// ---- POUs/Vorlagen/RFID/FB_RFID.TcPOU
FUNCTION_BLOCK FB_RFID
VAR_INPUT
	PermissionHardware	:	BOOL;	//Freigabe Hardware
	QuitError	:	BOOL;	//Fehler quittieren
	Reset	:	BOOL;	//Reset Commands
	SensorPartDetected	:	BOOL;	//Sensor Teil erkannt
	CommandID	:	WORD;	//Wird nach einem Befehl immer um 1 erhoeht
	ReadData	:	WORD;	//Gelesener Wert an der Stelle vom MemoryIndex
	Status	:	WORD;	//Status ungleich 0 = Fehler
	ActorInstanceIndex	:	INT;	//Index in DropDown HMI
	ActorInstanceName	:	STRING;		//Name of the instance
END_VAR
VAR_OUTPUT
	ExecuteCommand	:	BOOL;
	FMReadingSerialNumber	:	BOOL;	//Fertigmeldung Lesen Seriennummer
	FMReadingData	:	BOOL;	//Fertigmeldung Lesen
	FMWritingData	:	BOOL;	//Fertigmeldung Schreiben
	Error	:	BOOL;	//Fehler
	ErrorID	:	WORD;	//Fehler-ID
	Command	:	WORD;	//Command-ID:
	WriteData	:	WORD;	//Daten die geschrieben werden
	MemoryIndex	:	WORD;	//Angewaehlten Memory-Index der gelesen/geschrieben werden soll
	ReadDataTag	:	ARRAY[0..127] OF WORD;	//Array mit allen gelesenen Daten
END_VAR
VAR_IN_OUT
	HMIInterface	:	MachineSectionHMIInterface;	//HMI-Interface
END_VAR
VAR
	statReadingSerialNumber	:	BOOL;
	statExecuteCommand	:	BOOL;
	statReadingData	:	BOOL;
	statWritingData	:	BOOL;
	statErrorActive	:	BOOL;
	statReadingSerialnumberFinished	:	BOOL;
	statReadingDataFinished	:	BOOL;
	statWritingDataFinished	:	BOOL;
	statSelectedCommand	:	WORD;
	statErrorID	:	WORD;
	statLastCommandID	:	WORD;
	statReadSerialNumber	:	WORD;
	statDataToWrite	:	WORD;
	statSelectedMemoryIndex	:	WORD;
	statReadDataCompelete	:	ARRAY[0..127] OF WORD;
	statCompleteDataToWrite	:	ARRAY[0..127] OF WORD;
	statStateReadSerialNumber	:	RFIDReadSerialnumberStates;
	statStateWriteData	:	RFIDReadWriteDataStates;
	statStateReadData	:	RFIDReadWriteDataStates;
	statRisingEdgeNewOrder	:	R_TRIG;
	statTONDelayWritting	:	TON;
	statTONDelayReading	:	TON;
	debugStepMemory	:	INT;
	
	internHMIInterface	:	MachineSectionHMIInterface;
	internRisingEdgeExecuteCommand	:	R_TRIG;
	internRisingEdgeReadAllDataFinished	:	R_TRIG;
END_VAR
VAR CONSTANT
	NOCOMMAND	:	WORD := 0;
	READSERIALNUMBERCOMMAND	:	WORD := 1;
	READDATACOMMAND	:	WORD := 2;
	WRITEDATACOMMAND	:	WORD := 3;
	CLEARALLDATACOMMAND	:	WORD := 4;
END_VAR

(*===================== HMI INTERFACE =====================*)
internHMIInterface := HMIInterface;

IF internHMIInterface.ActiveMachineSection = MachineSection.RFID AND
	internHMIInterface.SelectedActor = ActorInstanceIndex THEN
	(*===================== Status-Interface =====================*)
	internHMIInterface.RFID.RFIDStatus.PermissionHardware := PermissionHardware;
	internHMIInterface.RFID.RFIDStatus.PartPresent := SensorPartDetected;
	internHMIInterface.RFID.RFIDStatus.ErrorActive := statErrorActive;
	internHMIInterface.RFID.RFIDStatus.FMReading := statReadingDataFinished OR statReadingSerialnumberFinished;
	internHMIInterface.RFID.RFIDStatus.FMWritting := statWritingDataFinished;
	(*===================== Data-Interface =====================*)
	internHMIInterface.RFID.RFIDData.AllReadData := statReadDataCompelete; 
	IF internRisingEdgeReadAllDataFinished.Q THEN
		internHMIInterface.RFID.RFIDData.AllWriteData := statReadDataCompelete;
	END_IF
	(*===================== Execute Command =====================*)
	internRisingEdgeExecuteCommand(CLK := internHMIInterface.RFID.RFIDControl.ExecuteCommand);
	IF internRisingEdgeExecuteCommand.Q THEN
		CASE internHMIInterface.RFID.RFIDControl.SelectedCommand OF
			NOCOMMAND :
				statReadingSerialNumber := FALSE;
				statReadingData := FALSE;
				statWritingData := FALSE;
			READSERIALNUMBERCOMMAND:
				statReadingSerialNumber := TRUE;
			READDATACOMMAND:
				statReadingData := TRUE;
			WRITEDATACOMMAND:
				statCompleteDataToWrite := internHMIInterface.RFID.RFIDData.AllWriteData;
				statWritingData := TRUE;	
		END_CASE
	END_IF
	
	(*===================== Write Interface =====================*)
	HMIInterface := internHMIInterface;
END_IF

(*===================== Error Handling =====================*)
IF QuitError AND statErrorActive THEN
	statErrorActive := FALSE;
	statErrorID := 0;
END_IF
IF Status <> 0 THEN
	statErrorActive := TRUE;
	statErrorID := Status;
END_IF
IF PermissionHardware AND SensorPartDetected THEN
	(*===================== Reset Data =====================*)
	statRisingEdgeNewOrder(CLK:= statReadingSerialNumber OR statReadingData OR 
								 statWritingData);
	IF NOT SensorPartDetected OR statRisingEdgeNewOrder.Q
	THEN
		ResetData_On();
	ELSIF Reset THEN
		ResetData_On();
		statSelectedCommand := NOCOMMAND;
		statStateReadSerialNumber := RFIDReadSerialnumberStates.WAITINGTRIGGER;	
		statStateWriteData := RFIDReadWriteDataStates.WAITINGTRIGGER;
	END_IF
	IF CommandID = 0 AND statLastCommandID <> 0 THEN
		statLastCommandID := 0;
	END_IF
	(*===================== Read Serialnumber =====================*)
	CASE statStateReadSerialNumber OF
		RFIDReadSerialnumberStates.WAITINGTRIGGER :
		debugStepMemory := RFIDReadSerialnumberStates.WAITINGTRIGGER;
			IF statReadingSerialNumber THEN
				statReadingSerialNumber := FALSE;
				statStateReadSerialNumber := RFIDReadSerialnumberStates.SETTRIGGER;
			END_IF
		RFIDReadSerialnumberStates.SETTRIGGER:
			debugStepMemory := RFIDReadSerialnumberStates.SETTRIGGER;
			statExecuteCommand := TRUE;
			statSelectedCommand := READSERIALNUMBERCOMMAND;
			statStateReadSerialNumber := RFIDReadSerialnumberStates.WAITINGRESPONSE;
		RFIDReadSerialnumberStates.WAITINGRESPONSE:
			debugStepMemory := RFIDReadSerialnumberStates.WAITINGRESPONSE;
			IF statErrorActive THEN
				statStateReadSerialNumber := RFIDReadSerialnumberStates.ERRORACTIVE;
			ELSIF CommandID <> statLastCommandID THEN
				statStateReadSerialNumber := RFIDReadSerialnumberStates.RESPONSE;
				statExecuteCommand := FALSE;
				statSelectedCommand := NOCOMMAND;
			END_IF
		RFIDReadSerialnumberStates.RESPONSE:
			debugStepMemory := RFIDReadSerialnumberStates.RESPONSE;
			statReadSerialNumber := ReadData;
			statReadingSerialnumberFinished := TRUE;
			statStateReadSerialNumber := RFIDReadSerialnumberStates.WAITINGTRIGGER;
		RFIDReadSerialnumberStates.ERRORACTIVE:
			debugStepMemory := RFIDReadSerialnumberStates.ERRORACTIVE;
			IF NOT statErrorActive THEN
				statStateReadSerialNumber := RFIDReadSerialnumberStates.WAITINGTRIGGER;
			END_IF
	END_CASE;
	(*===================== Read Data =====================*)
	statTONDelayReading(IN:= statStateReadData = RFIDReadWriteDataStates.SETTRIGGER, 
						 PT:= T#100MS);
	CASE statStateReadData OF
		RFIDReadWriteDataStates.WAITINGTRIGGER :
		debugStepMemory := RFIDReadWriteDataStates.WAITINGTRIGGER;
			IF statReadingData THEN
				statReadingData := FALSE;
				statSelectedCommand := READDATACOMMAND;
				statSelectedMemoryIndex := 1;
				statStateReadData := RFIDReadWriteDataStates.SETTRIGGER;
			END_IF
		RFIDReadWriteDataStates.SETTRIGGER:
			debugStepMemory := RFIDReadWriteDataStates.SETTRIGGER;
			IF statTONDelayReading.Q THEN
				statExecuteCommand := TRUE;
				statStateReadData := RFIDReadWriteDataStates.WAITINGRESPONSE;
			END_IF
		RFIDReadWriteDataStates.WAITINGRESPONSE:
			debugStepMemory := RFIDReadWriteDataStates.WAITINGRESPONSE;
			IF statErrorActive THEN
				statStateReadData := RFIDReadWriteDataStates.ERRORACTIVE;
			ELSIF CommandID <> statLastCommandID THEN
				statStateReadData := RFIDReadWriteDataStates.RESPONSE;
 				statExecuteCommand := FALSE;
			END_IF
		RFIDReadWriteDataStates.RESPONSE:
			debugStepMemory := RFIDReadWriteDataStates.RESPONSE;
			statReadDataCompelete[statSelectedMemoryIndex -1] := ReadData;
			IF statSelectedMemoryIndex >= 127 THEN
				statStateReadData := RFIDReadWriteDataStates.FINISHED;	
			ELSE
				statSelectedMemoryIndex := statSelectedMemoryIndex + 1;
				statStateReadData := RFIDReadWriteDataStates.SETTRIGGER;	
			END_IF
		RFIDReadWriteDataStates.ERRORACTIVE:
			debugStepMemory := RFIDReadWriteDataStates.ERRORACTIVE;
			IF NOT statErrorActive THEN
				statStateReadData := RFIDReadWriteDataStates.WAITINGTRIGGER;
			END_IF
		RFIDReadWriteDataStates.FINISHED:
			statReadingDataFinished := TRUE;
			statSelectedCommand := NOCOMMAND;
			statStateReadData := RFIDReadWriteDataStates.WAITINGTRIGGER;
	END_CASE;
	internRisingEdgeReadAllDataFinished(CLK := statReadingDataFinished);
	(*===================== Write Data =====================*)
	statTONDelayWritting(IN:= statStateWriteData = RFIDReadWriteDataStates.SETTRIGGER, 
						 PT:= T#100MS);
	CASE statStateWriteData OF
		RFIDReadWriteDataStates.WAITINGTRIGGER :
		debugStepMemory := RFIDReadWriteDataStates.WAITINGTRIGGER;
			IF statWritingData THEN
				statWritingData := FALSE;
				statSelectedCommand := WRITEDATACOMMAND;
				statSelectedMemoryIndex := 1;
				statStateWriteData := RFIDReadWriteDataStates.SETTRIGGER;
			END_IF
		RFIDReadWriteDataStates.SETTRIGGER:
			debugStepMemory := RFIDReadWriteDataStates.SETTRIGGER;
			IF statTONDelayWritting.Q THEN
				statExecuteCommand := TRUE;
				statDataToWrite := statCompleteDataToWrite[statSelectedMemoryIndex - 1];
				statStateWriteData := RFIDReadWriteDataStates.WAITINGRESPONSE;
			END_IF
		RFIDReadWriteDataStates.WAITINGRESPONSE:
			debugStepMemory := RFIDReadWriteDataStates.WAITINGRESPONSE;
			IF statErrorActive THEN
				statStateWriteData := RFIDReadWriteDataStates.ERRORACTIVE;
			ELSIF CommandID <> statLastCommandID THEN
				statStateWriteData := RFIDReadWriteDataStates.RESPONSE;
 				statExecuteCommand := FALSE;
			END_IF
		RFIDReadWriteDataStates.RESPONSE:
			debugStepMemory := RFIDReadWriteDataStates.RESPONSE;
			IF statSelectedMemoryIndex >= 127 THEN
				statStateWriteData := RFIDReadWriteDataStates.FINISHED;	
			ELSE
				statSelectedMemoryIndex := statSelectedMemoryIndex + 1;
				statStateWriteData := RFIDReadWriteDataStates.SETTRIGGER;	
			END_IF
		RFIDReadWriteDataStates.ERRORACTIVE:
			debugStepMemory := RFIDReadWriteDataStates.ERRORACTIVE;
			IF NOT statErrorActive THEN
				statStateWriteData := RFIDReadWriteDataStates.WAITINGTRIGGER;
			END_IF
		RFIDReadWriteDataStates.FINISHED:
			statWritingDataFinished := TRUE;
			statSelectedCommand := NOCOMMAND;
			statStateWriteData := RFIDReadWriteDataStates.WAITINGTRIGGER;
	END_CASE;
	(*===================== Save Data =====================*)
	statLastCommandID := CommandID;
ELSE
	statReadingSerialNumber := FALSE;	
	statReadingData := FALSE;
	statWritingData := FALSE;
	statExecuteCommand := FALSE;
	statReadingSerialnumberFinished := FALSE;
	statReadingDataFinished := FALSE;
	statWritingDataFinished := FALSE;
	statSelectedCommand := NOCOMMAND;
END_IF
(*===================== Outputs =====================*)
ExecuteCommand := statExecuteCommand;
FMReadingSerialNumber := statReadingSerialnumberFinished;
FMReadingData := statReadingDataFinished;
FMWritingData := statWritingDataFinished;
Error := statErrorActive;
ErrorID := statErrorID;
Command := statSelectedCommand;
WriteData := statDataToWrite;
MemoryIndex := statSelectedMemoryIndex;
ReadDataTag := statReadDataCompelete;

METHOD PUBLIC ReadDataComplete : BOOL
VAR_INPUT
	StartReadData	:	BOOL;
END_VAR
IF StartReadData THEN
	statReadingData := TRUE;
	ReadDataComplete := TRUE;
ELSE
	ReadDataComplete := FALSE;
END_IF
END_METHOD

METHOD PUBLIC ReadSerialNumber : BOOL
VAR_INPUT
	Start_ReadingSerialNumebr	:	BOOL;
END_VAR
IF Start_ReadingSerialNumebr AND NOT statErrorActive AND
	SensorPartDetected
THEN
	statReadingSerialNumber := TRUE;
	ReadSerialNumber := TRUE;
ELSE
	ReadSerialNumber := FALSE;			
END_IF
END_METHOD

METHOD PRIVATE ResetData_On : BOOL
VAR
	i :	INT;	//Laufvariable abloeschen gelesene Daten
END_VAR
statReadingSerialnumberFinished := FALSE;
statReadingDataFinished := FALSE;
statWritingDataFinished := FALSE;
statExecuteCommand := FALSE;
statReadSerialNumber := 0;
statDataToWrite := 0;
statSelectedMemoryIndex := 0;
statSelectedCommand := NOCOMMAND;
FOR i := 0 TO 127 DO
	statReadDataCompelete[i] := 0;
END_FOR

ResetData_On := TRUE;
END_METHOD

METHOD WriteDataComplete : BOOL
VAR_INPUT
	StartWriteData	:	BOOL;
	CompleteDataToWrite	:	ARRAY [0..127] OF WORD;
END_VAR
IF StartWriteData THEN
	statWritingData := TRUE;
	statCompleteDataToWrite := CompleteDataToWrite;	
	WriteDataComplete := TRUE;
ELSE
	WriteDataComplete := FALSE;
END_IF
END_METHOD

END_FUNCTION_BLOCK

// ---- POUs/Vorlagen/VisionSensor/FB_VisionSensor.TcPOU
FUNCTION_BLOCK FB_VisionSensor
VAR_INPUT
	PartPresent	:	BOOL;	//Part is on VisionSensor
	ValueCode	:	WORD;	//Material Code, which is detected
END_VAR
VAR_OUTPUT
	Finished	:	BOOL;	//Evaluation finished
	Error	:	BOOL;	//Error by evaluation of material
END_VAR
VAR
	statDetectedPart	:	VisionSensorParttype;
	statREPartDetected	:	R_TRIG;	
	statPartPresentDelay	:	TON:=(PT := T#100ms);
	statResultEvaluation	:	BOOL;
	statEvaluationFinished	:	BOOL;
	statErrorDetection	:	BOOL;
END_VAR

statPartPresentDelay(IN := PartPresent);
statREPartDetected(CLK := statPartPresentDelay.Q);
IF statREPartDetected.Q THEN
	statEvaluationFinished := FALSE;
	statResultEvaluation := GetParttype(ValueCode);
	IF statResultEvaluation THEN
		statEvaluationFinished := TRUE;
		statErrorDetection := FALSE;	
	ELSE
		statEvaluationFinished := TRUE;
		statErrorDetection := TRUE;				
	END_IF
ELSIF NOT PartPresent AND statDetectedPart <> VisionSensorParttype.None THEN
	statDetectedPart := VisionSensorParttype.None;
	statEvaluationFinished := FALSE;
	statResultEvaluation := FALSE;
	statErrorDetection := FALSE;
END_IF

Finished := statEvaluationFinished;
Error := statErrorDetection;

METHOD PRIVATE GetParttype : BOOL
VAR_INPUT
	valueCode	:	WORD;
END_VAR
VAR
	tempEvaluationSuccessfully	:	BOOL := FALSE;
	tempEvaluatedCode	:	VisionSensorParttype;
END_VAR
CASE valueCode OF
	VisionSensorParttype.None:
		tempEvaluatedCode := VisionSensorParttype.None;
		tempEvaluationSuccessfully := TRUE;
	VisionSensorParttype.BlueRawMaterial:
		tempEvaluatedCode := VisionSensorParttype.BlueRawMaterial;
		tempEvaluationSuccessfully := TRUE;
	VisionSensorParttype.BlueProductLid:
		tempEvaluatedCode := VisionSensorParttype.BlueProductLid;
		tempEvaluationSuccessfully := TRUE;
	VisionSensorParttype.BlueProductBase:
		tempEvaluatedCode := VisionSensorParttype.BlueProductBase;
		tempEvaluationSuccessfully := TRUE;
	VisionSensorParttype.GreenRawMaterial:
		tempEvaluatedCode := VisionSensorParttype.GreenRawMaterial;
		tempEvaluationSuccessfully := TRUE;
	VisionSensorParttype.GreenProductLid:
		tempEvaluatedCode := VisionSensorParttype.GreenProductLid;
		tempEvaluationSuccessfully := TRUE;
	VisionSensorParttype.GreenProductBase:
		tempEvaluatedCode := VisionSensorParttype.GreenProductBase;
		tempEvaluationSuccessfully := TRUE;
	VisionSensorParttype.MetalRawMaterial:
		tempEvaluatedCode := VisionSensorParttype.MetalRawMaterial;
		tempEvaluationSuccessfully := TRUE;
	VisionSensorParttype.MetalProductLid:
		tempEvaluatedCode := VisionSensorParttype.MetalProductLid;
		tempEvaluationSuccessfully := TRUE;
	VisionSensorParttype.MetalProductBase:
		tempEvaluatedCode := VisionSensorParttype.MetalProductBase;
		tempEvaluationSuccessfully := TRUE;
	ELSE
		tempEvaluatedCode := VisionSensorParttype.NotDectedable;
		tempEvaluationSuccessfully := FALSE;
END_CASE

statDetectedPart := tempEvaluatedCode;
GetParttype := tempEvaluationSuccessfully;
END_METHOD

PROPERTY PUBLIC Parttype : VisionSensorParttype
GET
Parttype := statDetectedPart;
END_GET
END_PROPERTY

END_FUNCTION_BLOCK

// ---- POUs/Vorlagen/Warehouse/FB_StackerCrane_Numerical.TcPOU
FUNCTION_BLOCK FB_StackerCrane_Numerical
VAR_INPUT
	XAxisMoving	:	BOOL;	//X axis is moving
	ZAxisMoving	:	BOOL;	//Z axis is moving
	ForkInPosLeft	:	BOOL;	//Fork is in the left position
	ForkInPosMiddle	:	BOOL;	//Fork is in the middle position
	ForkInPosRight	:	BOOL;	//Fork is in the right position
	ActorInstanceIndex	:	INT;	//Index in DropDown HMI
	ActorInstanceName	:	STRING;		//Name of the instance
END_VAR
VAR_OUTPUT
	LiftFork	:	BOOL;	//TRUE: Lift fork on current pos, FALSE: Lower fork on current pos, 
	MoveForkLeft	:	BOOL;	//Move Fork to the left pos
	MoveForkRight	:	BOOL;	//Move Fork to the right pos
	TargetPos	:	WORD;	//TargetPos for stacker crane
END_VAR
VAR_IN_OUT
	OperatingMode	:	OperatingMode;	//Schnittstelle für Betriebsarten
	HMIInterface	:	MachineSectionHMIInterface;	//HMI-Interface
END_VAR
VAR
	statMoveStackerCrane	:	BOOL;
	statStackerCraneNewOrder	:	BOOL;
	statStackerCraneInPositionXAxis	:	BOOL := TRUE;
	statStackerCraneInPositionZAxis	:	BOOL := TRUE;
	statMoveForkLeft	:	BOOL;
	statMoveForkRight	:	BOOL;
	statLiftFork	:	BOOL;
	statSelectedTargetPos	: WORD;
	statPropTargetPos	:	WORD := 55;
	statREXAxisMoving	:	R_TRIG;
	statREZAxisMoving	:	R_TRIG;
	statFEXAxisMoving	:	F_TRIG;
	statFEZAxisMoving	:	F_TRIG;
	
	internHMIInterface	:	MachineSectionHMIInterface;
	internInstanceActivatedFirstTime	:	BOOL;
	internRisingEdgePressButtonConfirm	:	R_TRIG;
	internRisingEdgePressButtonMove	:	R_TRIG;
	internRisingEdgePressButtonForkLift	:	R_TRIG;
	internRisingEdgePressButtonForkLower	:	R_TRIG;
	internRisingEdgePressButtonForkLeft	:	R_TRIG;
	internRisingEdgePressButtonForkRight	:	R_TRIG;
	internRisingEdgePressButtonMiddleFork	:	R_TRIG;
	internMiddleFork	:	BOOL;
END_VAR

(*===================== HMI INTERFACE =====================*)
internHMIInterface := HMIInterface;

IF internHMIInterface.ActiveMachineSection = MachineSection.StackerCrane AND
	internHMIInterface.SelectedActor = ActorInstanceIndex THEN
	(*===================== Initializing HMI-Interface =====================*)
	IF NOT internInstanceActivatedFirstTime THEN
		FC_InitializingSettingLines(HMIInterface := internHMIInterface);
		internInstanceActivatedFirstTime := TRUE;
	END_IF
	(*===================== Button Handling Movement =====================*)
	internHMIInterface.Movements.NumericalInput.CaptionNumericalInput := 'Stacker Crane Target POS';
	internHMIInterface.Movements.NumericalInput.IsVisibleNumericalInput := TRUE;
	
	internHMIInterface.Movements.NumericalInput.ButtonsNumericalInput[1].IsVisibleButton := TRUE;
	internHMIInterface.Movements.NumericalInput.ButtonsNumericalInput[1].IsEnabled := OperatingMode.ManuelIsActive AND NOT
									 														OperatingMode.EStop.IsActive AND NOT
																							OperatingMode.Fault.IsActive AND NOT
																							statMoveStackerCrane;
	internHMIInterface.Movements.NumericalInput.ButtonsNumericalInput[1].InPosition := FALSE;
	internHMIInterface.Movements.NumericalInput.ButtonsNumericalInput[1].CaptionButton := 'Confirm';
	internHMIInterface.Movements.NumericalInput.ButtonsNumericalInput[1].PathImageButton := 'Images\ForwardConveyor.svg';
	
	internHMIInterface.Movements.NumericalInput.ButtonsNumericalInput[2].IsVisibleButton := TRUE;
	internHMIInterface.Movements.NumericalInput.ButtonsNumericalInput[2].IsEnabled := OperatingMode.ManuelIsActive;
	internHMIInterface.Movements.NumericalInput.ButtonsNumericalInput[2].InPosition := FALSE;
	internHMIInterface.Movements.NumericalInput.ButtonsNumericalInput[2].CaptionButton := 'Move';
	internHMIInterface.Movements.NumericalInput.ButtonsNumericalInput[2].PathImageButton := 'Images\StopConveyor.svg';
	
	internHMIInterface.Movements.NumericalInput.ValueLinesNumericalInput[1].CaptionDescription := 'Selected Pos:';
	internHMIInterface.Movements.NumericalInput.ValueLinesNumericalInput[1].UnitInput := 'Storage Place';
	internHMIInterface.Movements.NumericalInput.ValueLinesNumericalInput[1].IsEnabledInput := TRUE;
	
	internHMIInterface.Movements.NumericalInput.ValueLinesNumericalInput[2].CaptionDescription := 'Current Pos:';
	internHMIInterface.Movements.NumericalInput.ValueLinesNumericalInput[2].UnitInput := 'Storage Place';
	internHMIInterface.Movements.NumericalInput.ValueLinesNumericalInput[2].ValueInput := statSelectedTargetPos;
	internHMIInterface.Movements.NumericalInput.ValueLinesNumericalInput[2].IsEnabledInput := FALSE;
	
	internHMIInterface.Movements.MovementSettingLines[2].CaptionSettingLine := CONCAT('StackerCrane Lift function ', ActorInstanceName);
	internHMIInterface.Movements.MovementSettingLines[2].VisibilitySettingLine := TRUE;
	
	internHMIInterface.Movements.MovementSettingLines[2].SettingLineButtons[1].IsVisibleButton := TRUE;
	internHMIInterface.Movements.MovementSettingLines[2].SettingLineButtons[1].IsVisibleAxisPosition := FALSE;
	internHMIInterface.Movements.MovementSettingLines[2].SettingLineButtons[1].IsEnabled := OperatingMode.ManuelIsActive AND NOT
									 														OperatingMode.EStop.IsActive AND NOT
																							OperatingMode.Fault.IsActive AND NOT
																							statMoveStackerCrane;
	internHMIInterface.Movements.MovementSettingLines[2].SettingLineButtons[1].InPosition := FALSE;
	internHMIInterface.Movements.MovementSettingLines[2].SettingLineButtons[1].CaptionButton := 'Lift';
	internHMIInterface.Movements.MovementSettingLines[2].SettingLineButtons[1].PathImageButton := 'Images\UpElevator.svg';
	
	internHMIInterface.Movements.MovementSettingLines[2].SettingLineButtons[2].IsVisibleButton := TRUE;
	internHMIInterface.Movements.MovementSettingLines[2].SettingLineButtons[2].IsVisibleAxisPosition := FALSE;
	internHMIInterface.Movements.MovementSettingLines[2].SettingLineButtons[2].IsEnabled := OperatingMode.ManuelIsActive AND NOT
									 														OperatingMode.EStop.IsActive AND NOT
																							OperatingMode.Fault.IsActive AND NOT
																							statMoveStackerCrane;
	internHMIInterface.Movements.MovementSettingLines[2].SettingLineButtons[2].InPosition := FALSE;
	internHMIInterface.Movements.MovementSettingLines[2].SettingLineButtons[2].CaptionButton := 'Lower';
	internHMIInterface.Movements.MovementSettingLines[2].SettingLineButtons[2].PathImageButton := 'Images\DownElevator.svg';
	
	internHMIInterface.Forks.ForkMovementSettingLines[1].CaptionSettingLine := CONCAT('Fork Control ', ActorInstanceName);
	internHMIInterface.Forks.ForkMovementSettingLines[1].VisibilitySettingLine := TRUE;
	
	internHMIInterface.Forks.ForkMovementSettingLines[1].SettingLineButtons[1].IsVisibleButton := TRUE;
	internHMIInterface.Forks.ForkMovementSettingLines[1].SettingLineButtons[1].IsVisibleAxisPosition := FALSE;
	internHMIInterface.Forks.ForkMovementSettingLines[1].SettingLineButtons[1].IsEnabled := OperatingMode.ManuelIsActive AND NOT
									 														OperatingMode.EStop.IsActive AND NOT
																							OperatingMode.Fault.IsActive AND NOT
																							statMoveStackerCrane AND
																							statStackerCraneInPositionXAxis AND
																							statStackerCraneInPositionZAxis;
	internHMIInterface.Forks.ForkMovementSettingLines[1].SettingLineButtons[1].InPosition := statMoveForkLeft;
	internHMIInterface.Forks.ForkMovementSettingLines[1].SettingLineButtons[1].CaptionButton := 'Left';
	internHMIInterface.Forks.ForkMovementSettingLines[1].SettingLineButtons[1].PathImageButton := 'Images\BackwardConveyor.svg';
	
	internHMIInterface.Forks.ForkMovementSettingLines[1].SettingLineButtons[2].IsVisibleButton := TRUE;
	internHMIInterface.Forks.ForkMovementSettingLines[1].SettingLineButtons[2].IsVisibleAxisPosition := FALSE;
	internHMIInterface.Forks.ForkMovementSettingLines[1].SettingLineButtons[2].IsEnabled := OperatingMode.ManuelIsActive;
	internHMIInterface.Forks.ForkMovementSettingLines[1].SettingLineButtons[2].InPosition := NOT statMoveForkLeft AND NOT statMoveForkRight;
	internHMIInterface.Forks.ForkMovementSettingLines[1].SettingLineButtons[2].CaptionButton := 'Stop';
	internHMIInterface.Forks.ForkMovementSettingLines[1].SettingLineButtons[2].PathImageButton := 'Images\StopConveyor.svg';
	
	internHMIInterface.Forks.ForkMovementSettingLines[1].SettingLineButtons[3].IsVisibleButton := TRUE;
	internHMIInterface.Forks.ForkMovementSettingLines[1].SettingLineButtons[3].IsVisibleAxisPosition := FALSE;
	internHMIInterface.Forks.ForkMovementSettingLines[1].SettingLineButtons[3].IsEnabled := OperatingMode.ManuelIsActive AND NOT
									 														OperatingMode.EStop.IsActive AND NOT
																							OperatingMode.Fault.IsActive AND NOT
																							statMoveStackerCrane AND
																							statStackerCraneInPositionXAxis AND
																							statStackerCraneInPositionZAxis;
	internHMIInterface.Forks.ForkMovementSettingLines[1].SettingLineButtons[3].InPosition := statMoveForkRight;
	internHMIInterface.Forks.ForkMovementSettingLines[1].SettingLineButtons[3].CaptionButton := 'Right';
	internHMIInterface.Forks.ForkMovementSettingLines[1].SettingLineButtons[3].PathImageButton := 'Images\ForwardConveyor.svg';
	
	(*===================== Confirm =====================*)
	internRisingEdgePressButtonConfirm(CLK := internHMIInterface.Movements.NumericalInput.ButtonsNumericalInput[1].IsPressed);
	IF internRisingEdgePressButtonConfirm.Q THEN
		statPropTargetPos := REAL_TO_WORD(internHMIInterface.Movements.NumericalInput.ValueLinesNumericalInput[1].ValueInput);
	END_IF
	(*===================== Move =====================*)
	internRisingEdgePressButtonMove(CLK := internHMIInterface.Movements.NumericalInput.ButtonsNumericalInput[2].IsPressed);
	IF internRisingEdgePressButtonMove.Q THEN
		statMoveStackerCrane := TRUE;
		statStackerCraneNewOrder := TRUE;
	END_IF
	(*===================== Fork Lift =====================*)
	internRisingEdgePressButtonForkLift(CLK := internHMIInterface.Movements.MovementSettingLines[2].SettingLineButtons[1].IsPressed);
	IF internRisingEdgePressButtonForkLift.Q THEN
		statLiftFork := TRUE;
	END_IF
	(*===================== Fork Lower =====================*)
	internRisingEdgePressButtonForkLower(CLK := internHMIInterface.Movements.MovementSettingLines[2].SettingLineButtons[2].IsPressed);
	IF internRisingEdgePressButtonForkLower.Q THEN
		statLiftFork := FALSE;
	END_IF
	(*===================== Fork Left =====================*)
	internRisingEdgePressButtonForkLeft(CLK := internHMIInterface.Forks.ForkMovementSettingLines[1].SettingLineButtons[1].IsPressed);
	IF internRisingEdgePressButtonForkLeft.Q THEN
		statMoveForkLeft := TRUE;
	END_IF
	(*===================== Fork Right =====================*)
	internRisingEdgePressButtonForkRight(CLK := internHMIInterface.Forks.ForkMovementSettingLines[1].SettingLineButtons[3].IsPressed);
	IF internRisingEdgePressButtonForkRight.Q THEN
		statMoveForkRight := TRUE;
	END_IF
	(*===================== Fork Middle =====================*)
	internRisingEdgePressButtonMiddleFork(CLK := internHMIInterface.Forks.ForkMovementSettingLines[1].SettingLineButtons[2].IsPressed);
	IF internRisingEdgePressButtonMiddleFork.Q THEN
		statMoveForkLeft := FALSE;
		statMoveForkRight := FALSE;
	END_IF
	
	(*===================== Write Interface =====================*)
	HMIInterface := internHMIInterface;
ELSE
		internInstanceActivatedFirstTime := FALSE;
END_IF
(*===================== Stacker crane in Position =====================*)
statREXAxisMoving(CLK := XAxisMoving);
statFEXAxisMoving(CLK := XAxisMoving);
statREZAxisMoving(CLK := ZAxisMoving);
statFEZAxisMoving(CLK := ZAxisMoving);

IF statStackerCraneInPositionXAxis AND statStackerCraneInPositionZAxis AND
NOT statStackerCraneNewOrder
THEN
	statMoveStackerCrane := FALSE;
END_IF
IF statREXAxisMoving.Q THEN
	statStackerCraneInPositionXAxis := FALSE;
	statStackerCraneNewOrder := FALSE;
END_IF
IF statFEXAxisMoving.Q THEN
	statStackerCraneInPositionXAxis := TRUE;
END_IF
IF statREZAxisMoving.Q THEN
	statStackerCraneInPositionZAxis := FALSE;
	statStackerCraneNewOrder := FALSE;
END_IF
IF statFEZAxisMoving.Q THEN
	statStackerCraneInPositionZAxis := TRUE;
END_IF 
(*===================== Positioning Stacker crane =====================*)
IF ((OperatingMode.AutomaticIsActive AND OperatingMode.AutomaticStart.IsActive) OR
	(OperatingMode.ManuelIsActive)) 
   AND statMoveStackerCrane 
THEN
	statSelectedTargetPos := statPropTargetPos;
// 	statStackerCraneNewOrder := FALSE;
END_IF
IF OperatingMode.EStop.IsActive OR OperatingMode.Fault.IsActive OR 
OperatingMode.AutomaticIsActive AND OperatingMode.AutomaticStop.IsActive
THEN
	statSelectedTargetPos := 0;
	statMoveStackerCrane := FALSE;
END_IF
(*===================== Outputs writting =====================*)
LiftFork := statLiftFork;
MoveForkLeft := statMoveForkLeft;
MoveForkRight := statMoveForkRight;
TargetPos := statSelectedTargetPos;

PROPERTY PUBLIC InPositionXAxis : BOOL
GET
InPositionXAxis := statStackerCraneInPositionXAxis;
END_GET
END_PROPERTY

PROPERTY PUBLIC InPositionZAxis : BOOL
GET
InPositionZAxis := statStackerCraneInPositionZAxis;
END_GET
END_PROPERTY

METHOD PUBLIC LiftForkUp : BOOL
VAR_INPUT
	StartLiftingFork	:	BOOL;
END_VAR
IF OperatingMode.AutomaticIsActive AND OperatingMode.AutomaticStart.IsActive AND
	InPositionXAxis AND InPositionZAxis AND StartLiftingFork AND NOT statMoveStackerCrane 
THEN
	statLiftFork := TRUE;
	LiftForkUp := TRUE;
ELSE
	LiftForkUp := FALSE;
END_IF
END_METHOD

METHOD PUBLIC LowerForkUp : BOOL
VAR_INPUT
	StartLoweringFork	:	BOOL;
END_VAR
IF OperatingMode.AutomaticIsActive AND OperatingMode.AutomaticStart.IsActive AND
	InPositionXAxis AND InPositionZAxis AND StartLoweringFork AND NOT statMoveStackerCrane 
THEN
	statLiftFork := FALSE;
	LowerForkUp := TRUE;
ELSE
	LowerForkUp := FALSE;
END_IF
END_METHOD

METHOD PUBLIC MoveAxesStackerCrane_ON : BOOL
VAR_INPUT
	StartMoveStackerCrane	:	BOOL;
	TargetPosStackerCrane	:	WORD;
END_VAR
IF OperatingMode.AutomaticIsActive AND OperatingMode.AutomaticStart.IsActive AND
	NOT statMoveStackerCrane AND StartMoveStackerCrane AND 
NumericalTargetPos <> TargetPosStackerCrane 
THEN
	NumericalTargetPos := TargetPosStackerCrane;
	statMoveStackerCrane := TRUE;
	statStackerCraneNewOrder := TRUE;
END_IF
END_METHOD

METHOD PUBLIC MoveForkToLeft_ON : BOOL
VAR_INPUT
	StartMovingForkLeft	:	BOOL;
END_VAR
IF OperatingMode.AutomaticIsActive AND OperatingMode.AutomaticStart.IsActive AND
	InPositionXAxis AND InPositionZAxis AND StartMovingForkLeft AND NOT statMoveStackerCrane 
THEN
	statMoveForkLeft := TRUE;
	MoveForkToLeft_ON := TRUE;
ELSE
	MoveForkToLeft_ON := FALSE;
END_IF
END_METHOD

METHOD PUBLIC MoveForkToMiddle_ON : BOOL
VAR_INPUT
	StartMovingForkMiddle: BOOL;
END_VAR
IF OperatingMode.AutomaticIsActive AND OperatingMode.AutomaticStart.IsActive AND 
	StartMovingForkMiddle THEN
	statMoveForkLeft := FALSE;
	statMoveForkRight := FALSE;
	MoveForkToMiddle_ON := TRUE;
ELSE
	MoveForkToMiddle_ON := FALSE;
END_IF
END_METHOD

METHOD PUBLIC MoveForkToRight_ON : BOOL
VAR_INPUT
	StartMovingForkRight	:	BOOL;
END_VAR
IF OperatingMode.AutomaticIsActive AND OperatingMode.AutomaticStart.IsActive AND
	InPositionXAxis AND InPositionZAxis AND StartMovingForkRight  AND NOT statMoveStackerCrane
THEN
	statMoveForkRight := TRUE;
	MoveForkToRight_ON := TRUE;
ELSE
	MoveForkToRight_ON := FALSE;
END_IF
END_METHOD

PROPERTY PUBLIC NewOrderActive : BOOL
GET
NewOrderActive := statStackerCraneNewOrder;
END_GET
SET
statStackerCraneNewOrder := NewOrderActive;
END_SET
END_PROPERTY

PROPERTY PUBLIC NumericalTargetPos : WORD
GET
NumericalTargetPos := statPropTargetPos;
END_GET
SET
IF NumericalTargetPos > 0 AND NumericalTargetPos < 56 THEN
	statPropTargetPos := NumericalTargetPos;
END_IF
END_SET
END_PROPERTY

END_FUNCTION_BLOCK

// ---- POUs/Vorlagen/OperatingMode/FB_OperatingMode.TcPOU
FUNCTION_BLOCK FB_OperatingMode
VAR_INPUT
	PermissionHardware	:	BOOL;	//Permission hardware ready for operation
	PermissionSoftware	:	BOOL;	//Permission from safety machine ready for start
	E_Stop	:	BOOL;	//Button E-Stop
	OperatingModeManual	:	BOOL;	//Operating Mode manual is selected
	OperatingModeAutomatic	:	BOOL;	//Operating Mode automatic is selected
END_VAR
VAR_OUTPUT
	LEDStart	:	BOOL;	//Indicator to show state automatic start
	LEDStop	:	BOOL;	//Indicator to show state automatic stop
	LEDHome	:	BOOL;	//Indicator to show state automatic home
	LEDReset	:	BOOL;	//Indicator to show state reset
	LEDQuit	:	BOOL;	//Indicator to show state quit
END_VAR
VAR_IN_OUT
	HMIInterface	:	HMIInterfaceOperatingMode;
END_VAR
VAR
	statRisingEdgeAutomaticActivated	:	BOOL;	//Rising edge, used when Automatic is activated
	statOperatingMode	:	OperatingMode;
	statHMIInterface	:	HMIInterfaceOperatingMode;
END_VAR

(*===================== Operating Manual =====================*)
statOperatingMode.ManuelIsActive := OperatingModeManual;
(*===================== Operating Automatic =====================*)
statOperatingMode.AutomaticIsActive := OperatingModeAutomatic;
(*===================== E-Stop is active =====================*)
statOperatingMode.EStop.PreconditionsFullfilled := TRUE;
statOperatingMode.EStop.IsActive := NOT E_Stop AND statOperatingMode.EStop.PreconditionsFullfilled;
(*===================== Reset is active =====================*)
statOperatingMode.Reset.PreconditionsFullfilled := TRUE;
statOperatingMode.Reset.IsActive := statOperatingMode.Reset.IsActive AND statOperatingMode.Reset.PreconditionsFullfilled;
(*===================== Quit is active =====================*)
statOperatingMode.Quit.PreconditionsFullfilled := TRUE;
statOperatingMode.Quit.IsActive := statOperatingMode.Quit.IsActive AND statOperatingMode.Quit.PreconditionsFullfilled;
(*===================== Automatic Start is active =====================*)
statOperatingMode.AutomaticStart.PreconditionsFullfilled := PermissionHardware AND PermissionSoftware AND
												  			E_Stop AND NOT statOperatingMode.Reset.IsActive AND NOT
												  			statOperatingMode.AutomaticHome.IsActive AND NOT
															statOperatingMode.Fault.IsActive AND
												  			statOperatingMode.AutomaticIsActive;
statOperatingMode.AutomaticStart.IsActive := statOperatingMode.AutomaticStart.IsActive AND statOperatingMode.AutomaticStart.PreconditionsFullfilled;
(*===================== Automatic Stop is active =====================*)
statOperatingMode.AutomaticStop.PreconditionsFullfilled := NOT statOperatingMode.AutomaticHome.IsActive;
statOperatingMode.AutomaticStop.IsActive := (statOperatingMode.AutomaticStop.IsActive AND statOperatingMode.AutomaticStop.PreconditionsFullfilled) OR
											 statOperatingMode.ManuelIsActive OR statOperatingMode.Fault.IsActive OR 
											 (statOperatingMode.AutomaticIsActive AND (NOT PermissionHardware OR NOT PermissionSoftware)) OR
											  statOperatingMode.EStop.IsActive OR statOperatingMode.Reset.IsActive;
IF statOperatingMode.AutomaticIsActive AND NOT statRisingEdgeAutomaticActivated THEN
	statRisingEdgeAutomaticActivated := TRUE;
	statOperatingMode.AutomaticStop.IsActive := TRUE;
ELSIF statOperatingMode.ManuelIsActive AND statRisingEdgeAutomaticActivated THEN
	statRisingEdgeAutomaticActivated := FALSE;
END_IF
(*===================== Automatic Home is active =====================*)
statOperatingMode.AutomaticHome.IsReached := statOperatingMode.AutomaticHome.AllMachinesInHome;
IF statOperatingMode.AutomaticHome.IsReached THEN
	StateOperatingMode.AutomaticStop.IsActive := TRUE;
END_IF
statOperatingMode.AutomaticHome.PreconditionsFullfilled := PermissionHardware AND PermissionSoftware AND
												  			E_Stop AND NOT statOperatingMode.Reset.IsActive AND
												  			statOperatingMode.AutomaticIsActive AND NOT
														   statOperatingMode.AutomaticHome.IsReached;
statOperatingMode.AutomaticHome.IsActive := statOperatingMode.AutomaticHome.IsActive AND statOperatingMode.AutomaticHome.PreconditionsFullfilled;
(*===================== Outputs =====================*)
LEDStart := statOperatingMode.AutomaticStart.IsActive;
LEDStop := statOperatingMode.AutomaticStop.IsActive;	
LEDHome := statOperatingMode.AutomaticHome.IsActive;	
LEDReset := statOperatingMode.Reset.IsActive;
LEDQuit	:= statOperatingMode.Quit.IsActive;

METHOD Homeing_On
VAR_INPUT
	ButtonHome	:	BOOL;
END_VAR
IF ButtonHome AND statOperatingMode.AutomaticStart.PreconditionsFullfilled AND NOT 
statOperatingMode.AutomaticHome.IsReached
THEN
	statOperatingMode.AutomaticStart.IsActive := FALSE;
	statOperatingMode.AutomaticStop.IsActive := FALSE;
	statOperatingMode.AutomaticHome.IsActive := TRUE;
END_IF
END_METHOD

METHOD PUBLIC Quit_On
VAR_INPUT
	ButtonQuit	:	BOOL;
END_VAR
IF ButtonQuit THEN
	statOperatingMode.Quit.IsActive := TRUE;
ELSE
		statOperatingMode.Quit.IsActive := FALSE;
END_IF
END_METHOD

METHOD PUBLIC Reset_on
VAR_INPUT
	ButtonReset	:	BOOL;
END_VAR
IF ButtonReset THEN
	statOperatingMode.Reset.IsActive := TRUE;
ELSE
		statOperatingMode.Reset.IsActive := FALSE;
END_IF
END_METHOD

METHOD PUBLIC Start_On
VAR_INPUT
	ButtonStart	:	BOOL;
END_VAR
IF ButtonStart AND statOperatingMode.AutomaticStart.PreconditionsFullfilled THEN
	statOperatingMode.AutomaticStart.IsActive := TRUE;
	statOperatingMode.AutomaticStop.IsActive := FALSE;
END_IF
END_METHOD

PROPERTY PUBLIC StateOperatingMode : REFERENCE TO OperatingMode
GET
StateOperatingMode REF= statOperatingMode;
END_GET
SET
statOperatingMode := StateOperatingMode;
END_SET
END_PROPERTY

METHOD PUBLIC Stop_On
VAR_INPUT
	ButtonStop	:	BOOL;
END_VAR
IF NOT ButtonStop AND statOperatingMode.AutomaticStart.PreconditionsFullfilled THEN
	statOperatingMode.AutomaticStart.IsActive := FALSE;
	statOperatingMode.AutomaticStop.IsActive := TRUE;
	statOperatingMode.AutomaticHome.IsActive := FALSE;
END_IF
END_METHOD

END_FUNCTION_BLOCK

// ---- POUs/Programm/ADS/Call_ADSCommunication.TcPOU
FUNCTION Call_ADSCommunication

RF_Data_Ready(CLK := instVisionSensorConveyor.Finished);

IF RF_Data_Ready.Q THEN
	Detected_Material := instVisionSensorConveyor.Parttype;
	Data_Ready := TRUE;
END_IF

END_FUNCTION

// ---- POUs/Programm/Aufzug/Call_Aufzug.TcPOU
FUNCTION Call_Aufzug

instFBElevator(
	CurrentPosition:= AufzugIstwert, 
	SensorOutfeed:= AufzugSensorAuslaufFoerderband, 
	SensorInfeed:= AufzugSensorEinlaufFoerderband, 
	ActorInstanceIndex := 0,
	ActorInstanceName := 'Zufuehrung',
	HMIInterface := HMI.hmiMachineSectionInterface,
	SetPointPositionElevator=> AufzugSollwert, 
	ConveyorForward=> AufzugFoerderbandVorwaerts, 
	ConveyorBackward=> AufzugFoerderbandRueckwaerts, 
	ElevatorInPosition=> AufzugInPosition, 
	OperatingMode:= instOperatingMode.StateOperatingMode);
	
instFBElevator.MoveElevator(AufzugBewegen, SollPosition);
instFBElevator.ConveyorForward_ON(AufzugFoerderbandVor);
instFBElevator.ConveyorBackward_ON(AufzugFoerderbandRueck);
instFBElevator.Conveyor_OFF(AufzugFoerderbandStop);

END_FUNCTION

// ---- POUs/Programm/Emitter/Call_Emitter.TcPOU
FUNCTION Call_Emitter
VAR_INPUT
END_VAR
VAR
END_VAR

instEmitter(PartPresent:= BauteilVorEmitter,
			ActorInstanceIndex := 0,
			ActorInstanceName := 'Zufuehrband',
			HMIInterface := HMI.hmiMachineSectionInterface, 
			CreatePart=> Emitter_Rollenband4m);
			
IF CreateNewPart THEN
	instEmitter.Create();
END_IF

IF BauteilVorEmitter THEN
	CreateNewPart := FALSE;
END_IF

END_FUNCTION

// ---- POUs/Programm/Foerderband/Call_Foerderband.TcPOU
FUNCTION Call_Foerderband

instFoerderband6(
	SensorInfeed:= Sensor_Band_Einlauf, 
	SensorOutfeed:= Sensor_Band_Auslauf, 
	MaximumTimeRuncontrol:= T#30S, 
	ActorInstanceIndex := 0,
	ActorInstanceName := 'Foerderband 6',
	HMIInterface := HMI.hmiMachineSectionInterface,
	MotorForward=> Foerderband_Vorwaerts, 
	MotorBackward=> Foerderband_Rueckwaerts, 
	RuncontrolForwardActive=> , 
	RuncontrolBackwardActive=> , 
	Error=> , 
	OperatingMode:= instOperatingMode.StateOperatingMode);

instFoerderband6.MotorForward_On(Sensor_Band_Einlauf OR StartButton);
instFoerderband6.MotorBackward_On(Sensor_Band_Auslauf);
instFoerderband6.Motor_Off((Foerderband_Vorwaerts AND Sensor_Band_Auslauf) OR
							(Foerderband_Rueckwaerts AND Sensor_Band_Einlauf));

END_FUNCTION

// ---- POUs/Programm/HMI/Call_HMI.TcPOU
FUNCTION Call_HMI

//hmiOperatingmodeInterface.PLCToHMI.CurrentOperatingMode := instOperatingMode.StateOperatingMode;
hmiHeaderInstance(NameApplication := 'Hochregallager',
				  OperatingModeHMIInterface := hmiOperatingmodeInterface,
				  HeaderHMIInterface := hmiHeaderInterface);
			  
hmiAdsCommunicationInterfaceInstance(Timeout := T#1S,
									 TimeoutHMI := T#500ms,
									 LocalAdsPort := 851,
									 HeartbeatHMI := hmiAdsCommunicationInterface.HeartbeatHMI);
									 

hmiAdsCommunicationInterface.DeviceIpAddress := hmiAdsCommunicationInterfaceInstance.LocalIpAddress;
hmiAdsCommunicationInterface.LocalAMSNetId := hmiAdsCommunicationInterfaceInstance.LocalAMSNetId;
hmiAdsCommunicationInterface.HeartbeatPLC := hmiAdsCommunicationInterfaceInstance.PLCHeartbeatHMICommunication;
hmiAdsCommunicationInterface.RuntimeStatus := hmiAdsCommunicationInterfaceInstance.AdsState;

// FC_InitializingSettingLines(HMIInterface := HMI.hmiMachineSectionInterface);

END_FUNCTION

// ---- POUs/Programm/MAIN.TcPOU
PROGRAM MAIN
VAR
	
END_VAR

SignalmappingInput();
Call_HMI();
Call_Emitter();
Call_OperatingMode();
// Call_Foerderband();
Call_Aufzug();
Call_Warehouse();
Call_RFID();
Call_VisionSensor();
Call_ADSCommunication();
Call_PositingBar();
Call_PickPlace();
Call_Remover();
SignalmappingOutput();

END_PROGRAM

// ---- POUs/Programm/SignalmappingInput.TcPOU
FUNCTION SignalmappingInput

(* ==================================== Digitale Eingaenge ====================================*)
BauteilVorEmitter := GVL.mb_Output_Coils[0];
BetrMan := GVL.mb_Output_Coils[1];
BetrAuto := GVL.mb_Output_Coils[2];
StartButton := GVL.mb_Output_Coils[3];
StopButton := GVL.mb_Output_Coils[4];
HomeButton := GVL.mb_Output_Coils[5];
ResetButton := GVL.mb_Output_Coils[6];
QuitButton	:= GVL.mb_Output_Coils[7]; 
E_Stop := GVL.mb_Output_Coils[8];
Sensor_Band_Einlauf := GVL.mb_Output_Coils[9];
Sensor_Band_Auslauf := GVL.mb_Output_Coils[10];
AufzugSensorEinlaufFoerderband := GVL.mb_Output_Coils[11];
AufzugSensorAuslaufFoerderband := GVL.mb_Output_Coils[12];
RBGEndlageMitte := GVL.mb_Output_Coils[13];
RBGEndlageLinks := GVL.mb_Output_Coils[14];
RBGEndlageRechts := GVL.mb_Output_Coils[15];
PartDetectedVisionSensor := GVL.mb_Output_Coils[18];
DigitalStackerCraneEndlageLinks := GVL.mb_Output_Coils[20];
DigitalStackerCraneEndlageMitte := GVL.mb_Output_Coils[21];
DigitalStackerCraneEndlageRechts := GVL.mb_Output_Coils[22];
DigitalStackerCraneXAxisIsMoving := GVL.mb_Output_Coils[23];
DigitalStackerCraneZAxisIsMoving := GVL.mb_Output_Coils[24];
PositionerIsClamped	:=	GVL.mb_Output_Coils[26];
PositionerIsRaised	:=	GVL.mb_Output_Coils[27];
PickPlaceX_YAxisIsMoving	:=	GVL.mb_Output_Coils[29];
PickPlaceZAxisIsMoving	:=	GVL.mb_Output_Coils[30];
PickPlaceBoxDetected	:=	GVL.mb_Output_Coils[31];
PickPlaceCAxisInPos	:=	GVL.mb_Output_Coils[32];
RemoverPartPresent	:=	GVL.mb_Output_Coils[34];

(* ==================================== Analoge Eingaenge ====================================*)
AufzugIstwert := GVL.mb_Output_Registers[0];
RBGIstwertX := GVL.mb_Output_Registers[1];
RBGIstwertZ := GVL.mb_Output_Registers[2];
RFIDCommandID := GVL.mb_Output_Registers[3];
RFIDReadData := GVL.mb_Output_Registers[4];
RFIDStatus := GVL.mb_Output_Registers[5];
ReadPartCode := GVL.mb_Output_Registers[6];
PickPlacePositionXAxis	:=	GVL.mb_Output_Registers[9];
PickPlacePositionYAxis	:=	GVL.mb_Output_Registers[10];
PickPlacePositionZAxis	:=	GVL.mb_Output_Registers[11];

END_FUNCTION

// ---- POUs/Programm/OperatingMode/Call_OperatingMode.TcPOU
FUNCTION Call_OperatingMode

instOperatingMode(PermissionHardware:= simPermissionHardware, 
				  PermissionSoftware:= simPermissionSafety, 
				  E_Stop:= E_Stop, 
				  OperatingModeManual:= BetrMan, 
				  OperatingModeAutomatic:= BetrAuto,
				  HMIInterface :=  hmiOperatingmodeInterface,
				  LEDStart=> StartLED, 
				  LEDStop=> StopLED, 
				  LEDHome=> HomeLED, 
				  LEDReset=> ResetLED, 
				  LEDQuit=> QuitLED);

instOperatingMode.Start_On(StartButton);
instOperatingMode.Stop_On(StopButton);
instOperatingMode.Homeing_On(HomeButton);
instOperatingMode.Reset_On(ResetButton);
instOperatingMode.Quit_On(QuitButton);

END_FUNCTION

// ---- POUs/Programm/Warehouse/Call_Warehouse.TcPOU
FUNCTION Call_Warehouse
VAR
	iCounter	:	INT := -1;
END_VAR

// (*================ Analog Stacker crane ================*)
// instStackerCraneAnalog(StackerCraneCurrentPositionXAxis := RBGIstwertX,
//                  StackerCraneCurrentPositionZAxis := RBGIstwertZ,
// 				 ActorInstanceIndex := 0,
// 				 ActorInstanceName := 'Einlagerung',
// 				 HMIInterface := HMI.hmiMachineSectionInterface,
// 				 OperatingMode := instOperatingMode.StateOperatingMode,
// 				 SetPointToXAxis => RBGSollwertX, 
//                  SetPointToZAxis => RBGSollwertZ, 
//                  MoveForkLeft => RBGGabelLinks,	
//                  MoveForkRight => RBGGabelRechts);
// instStackerCraneAnalog.MoveAxesStackerCrane_ON(RBGStartMove, RBGSollwertXSimu, RBGSollwertZSimu);
// instStackerCraneAnalog.MoveForkToLeft_ON(RBGStartForkLeftMove);
// instStackerCraneAnalog.MoveForkToRight_ON(RBGStartForkRightMove);
// instStackerCraneAnalog.MoveForkToMiddle_ON(RBGStartForkMiddleMove);
// (*================ Steps ================*)
// IF instOperatingMode.StateOperatingMode.Reset.IsActive THEN
// 	processStepsAnalogStackerCrane := StackerCraneSteps.Waiting;
// END_IF
// 
// CASE processStepsAnalogStackerCrane OF
// 	StackerCraneSteps.Waiting:
// 		instStackerCraneAnalog.MoveForkToMiddle_ON(TRUE);
// 		IF instOperatingMode.StateOperatingMode.AutomaticStart.IsActive THEN
// 			processStepsAnalogStackerCrane := StackerCraneSteps.DriveToLoadingPosition;
// 		END_IF
// StackerCraneSteps.DriveToLoadingPosition:
// 		instStackerCraneAnalog.MoveAxesStackerCrane_ON(TRUE, 0.0, 0.0);
// 		instStackerCraneAnalog.EvaluatePosition();
// 		IF instStackerCraneAnalog.InPositionXAxis AND instStackerCraneAnalog.InPositionZAxis   
// 		AND TRUE
// 		THEN
// 			InUnloadingAnalog	:= FALSE;
// 			processStepsAnalogStackerCrane := StackerCraneSteps.ForkUnderLoad;
// 		END_IF
// StackerCraneSteps.ForkUnderLoad:
// 		InUnloadingAnalog	:= FALSE;
// 		instStackerCraneAnalog.MoveForkToLeft_ON(TRUE);
// 		IF RBGEndlageLinks THEN
// 			processStepsAnalogStackerCrane := StackerCraneSteps.LiftLoadItem;
// 		END_IF
// StackerCraneSteps.LiftLoadItem:
// 		instStackerCraneAnalog.MoveForkToLeft_ON(TRUE);
// 		instStackerCraneAnalog.MoveAxesStackerCrane_ON(TRUE, 0.0, 1.0);
// 		instStackerCraneAnalog.EvaluatePosition();
// 		IF instStackerCraneAnalog.InPositionXAxis AND instStackerCraneAnalog.InPositionZAxis 
// 		AND TRUE
// 		THEN
// 			processStepsAnalogStackerCrane := StackerCraneSteps.ForkToMiddle;
// 		END_IF
// StackerCraneSteps.ForkToMiddle:
// 		instStackerCraneAnalog.MoveForkToMiddle_ON(TRUE);
// 		IF RBGEndlageMitte AND NOT InUnloadingAnalog THEN
// 			processStepsAnalogStackerCrane := StackerCraneSteps.DriveToUnloadPrePosition;
// 		ELSIF RBGEndlageMitte AND InUnloadingAnalog THEN
// 			processStepsAnalogStackerCrane := StackerCraneSteps.DriveToLoadingPosition;
// 		END_IF
// StackerCraneSteps.DriveToUnloadPrePosition:
// 		instStackerCraneAnalog.MoveAxesStackerCrane_ON(TRUE, 1.10, 1.86);
// 		instStackerCraneAnalog.EvaluatePosition();
// 		IF instStackerCraneAnalog.InPositionXAxis AND instStackerCraneAnalog.InPositionZAxis   
// 		AND TRUE
// 		THEN
// 			processStepsAnalogStackerCrane := StackerCraneSteps.ForkInWarehouse;
// 		END_IF
// StackerCraneSteps.ForkInWarehouse:
// 		instStackerCraneAnalog.MoveForkToRight_ON(TRUE);
// 		IF RBGEndlageRechts THEN
// 			processStepsAnalogStackerCrane := StackerCraneSteps.DriveToUnloadPosition;
// 		END_IF
// StackerCraneSteps.DriveToUnloadPosition:
// 		instStackerCraneAnalog.MoveForkToRight_ON(TRUE);
// 		instStackerCraneAnalog.MoveAxesStackerCrane_ON(TRUE, 1.15, 1.26);
// 		instStackerCraneAnalog.EvaluatePosition();
// 		IF instStackerCraneAnalog.InPositionXAxis AND instStackerCraneAnalog.InPositionZAxis  
// 		AND TRUE
// 		THEN
// 			InUnloadingAnalog	:= TRUE;
// 			processStepsAnalogStackerCrane := StackerCraneSteps.ForkToMiddle;
// 		END_IF
// END_CASE


(*================ Numerical Stacker crane ================*)
instStackerCraneNumerical(XAxisMoving := DigitalStackerCraneXAxisIsMoving,
						  ZAxisMoving := DigitalStackerCraneZAxisIsMoving,
						  ActorInstanceIndex := 1,
						  ActorInstanceName := 'Zufuehrung',
						  ForkInPosLeft := DigitalStackerCraneEndlageLinks,
						  ForkInPosMiddle := DigitalStackerCraneEndlageMitte,
						  ForkInPosRight := DigitalStackerCraneEndlageRechts,
						  OperatingMode := instOperatingMode.StateOperatingMode,
						  HMIInterface := HMI.hmiMachineSectionInterface,
						  LiftFork => DigitalStackerCraneLiftGabel,
						  MoveForkLeft => DigitalStackerCraneGabelLinks,
						  MoveForkRight => DigitalStackerCraneGabelRechts,
						  TargetPos => DigitalStackerCraneTargetPos);
// instStackerCraneNumerical.MoveAxesStackerCrane_ON(DigtalStackerCraneStartMove, DigitalTargetPosSimu);
// instStackerCraneNumerical.MoveForkToLeft_ON(DigtalStackerCraneStartForkLeftMove);
// instStackerCraneNumerical.MoveForkToRight_ON(DigtalStackerCraneStartForkRightMove);
// instStackerCraneNumerical.MoveForkToMiddle_ON(DigtalStackerCraneStartForkMiddleMove);						  
// instStackerCraneNumerical.LiftForkUp(DigitalStackerCraneStartLiftFork);
// instStackerCraneNumerical.LowerForkUp(NOT DigitalStackerCraneStartLiftFork);						  

(*================ Steps ================*)
IF instOperatingMode.StateOperatingMode.Reset.IsActive THEN
	processStepsNumericalStackerCrane := StackerCraneSteps.Waiting;
END_IF

CASE processStepsNumericalStackerCrane OF
	StackerCraneSteps.Waiting:
	iCounter := 0;
		instStackerCraneNumerical.MoveForkToMiddle_ON(TRUE);
		IF instOperatingMode.StateOperatingMode.AutomaticStart.IsActive THEN
			processStepsNumericalStackerCrane := StackerCraneSteps.DriveToLoadingPosition;
		END_IF
StackerCraneSteps.DriveToLoadingPosition:
		instStackerCraneNumerical.MoveAxesStackerCrane_ON(TRUE, 55);
		IF instStackerCraneNumerical.InPositionXAxis AND instStackerCraneNumerical.InPositionZAxis
			AND NOT instStackerCraneNumerical.NewOrderActive
		THEN
 			InUnloadingNumerical	:= FALSE;
			processStepsNumericalStackerCrane := StackerCraneSteps.ForkUnderLoad;
		END_IF
StackerCraneSteps.ForkUnderLoad:
		instStackerCraneNumerical.MoveForkToRight_ON(TRUE);
		IF DigitalStackerCraneEndlageRechts THEN
			processStepsNumericalStackerCrane := StackerCraneSteps.LiftLoadItem;
		END_IF
StackerCraneSteps.LiftLoadItem:
		instStackerCraneNumerical.MoveForkToRight_ON(TRUE);
		instStackerCraneNumerical.LiftForkUp(TRUE);
		IF instStackerCraneNumerical.InPositionXAxis AND instStackerCraneNumerical.InPositionZAxis
			AND Lifting
		THEN
			processStepsNumericalStackerCrane := StackerCraneSteps.ForkToMiddle;
		END_IF
		Lifting := TRUE;
StackerCraneSteps.ForkToMiddle:
		Lifting := FALSE;
		Lowering := FALSE;
		instStackerCraneNumerical.MoveForkToMiddle_ON(TRUE);
		IF DigitalStackerCraneEndlageMitte AND NOT InUnloadingNumerical THEN
			processStepsNumericalStackerCrane := StackerCraneSteps.DriveToUnloadPrePosition;
		ELSIF DigitalStackerCraneEndlageMitte AND InUnloadingNumerical THEN
			processStepsNumericalStackerCrane := StackerCraneSteps.DriveToLoadingPosition;
		END_IF
StackerCraneSteps.DriveToUnloadPrePosition:
		instStackerCraneNumerical.MoveAxesStackerCrane_ON(TRUE, 7);
		IF instStackerCraneNumerical.InPositionXAxis AND instStackerCraneNumerical.InPositionZAxis
			AND NOT instStackerCraneNumerical.NewOrderActive
		THEN
			processStepsNumericalStackerCrane := StackerCraneSteps.ForkInWarehouse;
		END_IF
StackerCraneSteps.ForkInWarehouse:
		instStackerCraneNumerical.MoveForkToLeft_ON(TRUE);
		IF DigitalStackerCraneEndlageLinks THEN
			processStepsNumericalStackerCrane := StackerCraneSteps.DriveToUnloadPosition;
		END_IF
StackerCraneSteps.DriveToUnloadPosition:
		instStackerCraneNumerical.MoveForkToLeft_ON(TRUE);
		instStackerCraneNumerical.LowerForkUp(TRUE);
		IF instStackerCraneNumerical.InPositionXAxis AND instStackerCraneNumerical.InPositionZAxis
			AND Lowering
		THEN
			InUnloadingNumerical	:= TRUE;
			processStepsNumericalStackerCrane := StackerCraneSteps.ForkToMiddle;
		END_IF
		Lowering := TRUE;
END_CASE

END_FUNCTION

// ---- POUs/Programm/RFID/Call_RFID.TcPOU
FUNCTION Call_RFID
VAR
	tempCounter	:	INT;
END_VAR


instFBRFID(PermissionHardware := simPermissionHardware,
		   QuitError := instOperatingMode.StateOperatingMode.Quit.IsActive,
		   Reset := instOperatingMode.StateOperatingMode.Reset.IsActive,
		   SensorPartDetected := Sensor_Band_Einlauf,
		   CommandID := RFIDCommandID,
		   ReadData := RFIDReadData,
		   Status := RFIDStatus,
		   ActorInstanceIndex := 0,
		   ActorInstanceName := 'Zufuehrung Warehouse',
		   HMIInterface := HMI.hmiMachineSectionInterface,
		   ExecuteCommand => RFIDExecuteCommand,
		   Command => RFIDCommand,
		   WriteData => RFIDWriteData,
		   MemoryIndex => RFIDMemoryIndex,
		   ReadDataTag => RFIDCompleteDataToReadSimu);

FOR tempCounter := 0 TO 127 DO
	RFIDCompleteDataToWriteSimu[tempCounter] := tempCounter;
END_FOR		 
instFBRFID.ReadSerialNumber(RFIDReadSerialNumberSimu);
instFBRFID.WriteDataComplete(RFIDWriteDataSimu, RFIDCompleteDataToWriteSimu);
instFBRFID.ReadDataComplete(RFIDReadDataSimu);
IF RFIDReadSerialNumberSimu OR RFIDWriteDataSimu OR RFIDReadDataSimu THEN
	RFIDReadSerialNumberSimu := FALSE;
	RFIDWriteDataSimu := FALSE;
	RFIDReadDataSimu := FALSE;
END_IF

END_FUNCTION

// ---- POUs/Programm/VisionSensor/Call_VisionSensor.TcPOU
FUNCTION Call_VisionSensor

instVisionSensorConveyor(PartPresent := PartDetectedVisionSensor,
													ValueCode := ReadPartCode,
													Error => ErrorVisionSensor);

END_FUNCTION

// ---- POUs/Programm/PositingBar/Call_PositingBar.TcPOU
FUNCTION Call_PositingBar

instControlBlockPositingBar(PartIsClamped := PositionerIsClamped,
							VerticalLimitReached := PositionerIsRaised,
							AlignmentDirection	:= PositingBarAlignmentDirection.AlingmentLeft,
							ActorInstanceIndex := 1,
							ActorInstanceName := '',
							OperatingMode := instOperatingMode.StateOperatingMode,
							HMIInterface := HMI.hmiMachineSectionInterface,
							Clamp => PositionerClamp,
							Raise =>PositionerRaise);
							
IF SimuClampPositingBar THEN
	SimuUnclampPositingBar := FALSE;
END_IF
IF SimuUnclampPositingBar THEN
	SimuClampPositingBar := FALSE;
END_IF
IF SimuRaisePositingBar THEN
	SimuLowerPositingBar := FALSE;
END_IF
IF SimuLowerPositingBar THEN
	SimuRaisePositingBar := FALSE;
END_IF

instControlBlockPositingBar.PositingBarClamping(SimuClampPositingBar);
instControlBlockPositingBar.PositingBarUnclamping(SimuUnclampPositingBar);
instControlBlockPositingBar.PositingBarRaise(SimuRaisePositingBar);
instControlBlockPositingBar.PositingBarLower(SimuLowerPositingBar);

END_FUNCTION

// ---- POUs/Programm/PickPlace/Call_PickPlace.TcPOU
FUNCTION Call_PickPlace

instPickPlaceDigitalAnalog(
	PickPlaceCurrentPositionXAxis := PickPlacePositionXAxis,
	PickPlaceCurrentPositionYAxis := PickPlacePositionYAxis,
	PickPlaceCurrentPositionZAxis := PickPlacePositionZAxis,
	PickPlaceX_YAxisStillMoving := PickPlaceX_YAxisIsMoving,
	PickPlaceZAxisStillMoving := PickPlaceZAxisIsMoving,
	PickPlaceBoxDetected := PickPlaceBoxDetected,
	PickPlaceCAxisLimitReached := PickPlaceCAxisInPos,
	ActorInstanceIndex := 0,
	ActorInstanceName := 'Zufuehrband',
	OperatingMode := instOperatingMode.StateOperatingMode,
	HMIInterface := HMI.hmiMachineSectionInterface,
	SetPointToXAxis => PickPlaceSetpositionXAxis,
	SetPointToYAxis => PickPlaceSetpositionYAxis,
	SetPointToZAxis => PickPlaceSetpositionZAxis,
	GrabPart => PickPlaceGrabBox,
	RotateGripper => PickPlaceCAxisMovePlus);
	
	IF instOperatingMode.StateOperatingMode.Reset.IsActive THEN
			processStepsPickPlace := PickPlaceSteps.WaitingForAutomaticStart;
		END_IF
	WaitingTimeGrabPart(PT := T#2S);
	
	CASE processStepsPickPlace OF
		PickPlaceSteps.WaitingForAutomaticStart:
		
		IF instOperatingMode.StateOperatingMode.AutomaticStart.IsActive THEN
			processStepsPickPlace := PickPlaceSteps.DriveToHome;
		END_IF
		
		PickPlaceSteps.DriveToHome:
		
		instPickPlaceDigitalAnalog.MoveXYAxis_On(TRUE, HomePosition);
		instPickPlaceDigitalAnalog.MoveZAxis_On(TRUE, HomePosition);
		instPickPlaceDigitalAnalog.ReleasePart(TRUE);
		instPickPlaceDigitalAnalog.RotateGripperTo0(TRUE);
		IF instPickPlaceDigitalAnalog.InPositionX_Y_Axis AND 
			instPickPlaceDigitalAnalog.InPositionZAxis AND
		NOT instPickPlaceDigitalAnalog.NewOrderActive
		THEN
			processStepsPickPlace := PickPlaceSteps.DriveXYToPick;
			DelayProcessStep := FALSE;
		END_IF
		
		PickPlaceSteps.DriveXYToPick:
		
		instPickPlaceDigitalAnalog.MoveXYAxis_On(TRUE, PickPlacePosition);
		IF instPickPlaceDigitalAnalog.InPositionX_Y_Axis AND
		NOT instPickPlaceDigitalAnalog.NewOrderActive
		THEN
			processStepsPickPlace := PickPlaceSteps.DriveZDown;
			DelayProcessStep := FALSE;
		END_IF
		
		PickPlaceSteps.DriveZDown:
		
		instPickPlaceDigitalAnalog.MoveZAxis_On(TRUE, PickPlacePosition);
		IF instPickPlaceDigitalAnalog.InPositionZAxis  AND
		NOT instPickPlaceDigitalAnalog.NewOrderActive
		THEN
			processStepsPickPlace := PickPlaceSteps.GrabPart;
			DelayProcessStep := FALSE;
		END_IF
		
		PickPlaceSteps.GrabPart:
		WaitingTimeGrabPart(IN := TRUE);
		instPickPlaceDigitalAnalog.GrabPart_ON(TRUE);
		instPickPlaceDigitalAnalog.RotateGripperTo90(TRUE);
		IF WaitingTimeGrabPart.Q THEN
			WaitingTimeGrabPart(IN := FALSE);
			processStepsPickPlace := PickPlaceSteps.DriveZUp;
			DelayProcessStep := FALSE;
		END_IF
		
		PickPlaceSteps.DriveZUp:
		
		instPickPlaceDigitalAnalog.MoveZAxis_On(TRUE, HomePosition);
		IF instPickPlaceDigitalAnalog.InPositionZAxis AND
		NOT instPickPlaceDigitalAnalog.NewOrderActive
		THEN
			processStepsPickPlace := PickPlaceSteps.WaitingForAutomaticStart;
			DelayProcessStep := FALSE;
		END_IF
	END_CASE

END_FUNCTION

// ---- POUs/Programm/Remover/Call_Remover.TcPOU
FUNCTION Call_Remover

instFBRemover(PartPresent := RemoverPartPresent,
			  ActorInstanceIndex := 1,
			  ActorInstanceName := 'Remover conveyor',
			  HMIInterface := HMI.hmiMachineSectionInterface,
			  RemovePart => Remover);

END_FUNCTION

// ---- POUs/Programm/SignalmappingOutput.TcPOU
FUNCTION SignalmappingOutput

(* ==================================== Digitale Ausgaenge ====================================*)
	
	GVL.mb_Input_Coils[0] := Emitter_Rollenband4m;
	GVL.mb_Input_Coils[3] := StartLED;
	GVL.mb_Input_Coils[4] := StopLED;
	GVL.mb_Input_Coils[5] := ResetLED;
	GVL.mb_Input_Coils[6] := HomeLED;
	GVL.mb_Input_Coils[7] := QuitLED;
	GVL.mb_Input_Coils[9] := Foerderband_Vorwaerts;
	GVL.mb_Input_Coils[10] := Foerderband_Rueckwaerts;
	GVL.mb_Input_Coils[11] := AufzugFoerderbandVorwaerts;
	GVL.mb_Input_Coils[12] := AufzugFoerderbandRueckwaerts;
	GVL.mb_Input_Coils[14] := RBGGabelLinks;
	GVL.mb_Input_Coils[15] := RBGGabelRechts;
	GVL.mb_Input_Coils[17] := RFIDExecuteCommand;
	GVL.mb_Input_Coils[20] := DigitalStackerCraneGabelLinks;
	GVL.mb_Input_Coils[21] := DigitalStackerCraneGabelRechts;
	GVL.mb_Input_Coils[22] := DigitalStackerCraneLiftGabel;
	GVL.mb_Input_Coils[26]	:=	PositionerClamp;
	GVL.mb_Input_Coils[27]	:=	PositionerRaise;
	GVL.mb_Input_Coils[29]	:=	PickPlaceCAxisMovePlus;
	GVL.mb_Input_Coils[30]	:=	PickPlaceGrabBox;
	GVL.mb_Input_Coils[34]	:=	Remover;


(* ==================================== Analoge Ausgaenge ====================================*)
	GVL.mb_Input_Registers[0] := AufzugSollwert;
	GVL.mb_Input_Registers[1] := RBGSollwertX;
	GVL.mb_Input_Registers[2] := RBGSollwertZ;
	GVL.mb_Input_Registers[3] := RFIDCommand;
	GVL.mb_Input_Registers[4] := RFIDWriteData;
	GVL.mb_Input_Registers[5] := RFIDMemoryIndex;
	GVL.mb_Input_Registers[7] := DigitalStackerCraneTargetPos;
	GVL.mb_Input_Registers[9]	:=	PickPlaceSetpositionXAxis;
	GVL.mb_Input_Registers[10]	:=	PickPlaceSetpositionYAxis;
	GVL.mb_Input_Registers[11]	:=	PickPlaceSetpositionZAxis;

END_FUNCTION
